Fanuc KAREL source: KB00066.KL

PROGRAM KB00066
%NOLOCKGROUP
VAR
  P1: STRING[80]
  P2: INTEGER
  P3: ARRAY[4] OF STRING[80]
  P4: ARRAY[4] OF BOOLEAN
  P5: ARRAY[4] OF BOOLEAN
  P6: INTEGER
  P7: INTEGER
  P8: INTEGER
  P9: INTEGER
BEGIN
  P1 = 'A'
  P2 = 1
  P6 = 1
  P7 = 1
  P8 = 1
  P9 = 1
  DISCTRL_FORM(P1, P2, P3, P4, P5, P6, P7, P8, P9)
END KB00066
